//| use case:
//| Three variables are specified for historical access. 
//| Every three seconds their values should be updated to data storage for one second long.
PROGRAM PRG_HA_MultipleNodes
VAR CONSTANT
	// These connection and namespace settings need to be adapted to the runtime environment
	cOpcUaServerUrl			: STRING(MAX_STRING_LENGTH) := 'opc.tcp://localhost:4840';
	cNamespaceUri			: STRING(MAX_STRING_LENGTH) := 'urn:BeckhoffAutomation:Ua:PLC1';
END_VAR
VAR
	// Variables for HistorcalAccess
	{attribute 'OPC.UA.DA' := '1'}
	nMyValue1 : INT;	
	{attribute 'OPC.UA.DA' := '1'}
	nMyValue2 : INT;
	{attribute 'OPC.UA.DA' := '1'}
	fMyValue3 : LREAL;
	
	// state machine declarations 
	nState					: INT;
	bStart					: BOOL;  		//Set True to start this sample.
	bSample					: BOOL;			//Set True to stop the sampling.
	bStop					: BOOL;			//Set True to close the connection afterwards.
	bError					: BOOL;
	nErrorID				: DWORD;
	fbTimer					: TON:=(PT:=T#3S);
	
	// Declarations for UA_Connect
	fbUAConnect				: UA_Connect;
	stSessionConnectInfo 	: ST_UASessionConnectInfo;
	nConnectionHdl			: DWORD;
	
	// Declarations for UA_GetNamespaceIndex
	fbUAGetNamespaceIndex	: UA_GetNamespaceIndex;
	nNamespaceIndex			: UINT;
	
	// Declarations for UA_HistoryUpdate
	fbHistoryUpdateNode1	: FB_HistoryUpdate_INT := (sNodeIdentifier := 'PRG_HA_MultipleNodes.nMyValue1');
	fbHistoryUpdateNode2	: FB_HistoryUpdate_INT := (sNodeIdentifier := 'PRG_HA_MultipleNodes.nMyValue2');
	fbHistoryUpdateNode3	: FB_HistoryUpdate_LREAL := (sNodeIdentifier := 'PRG_HA_MultipleNodes.fMyValue3');
	
	// Declarations for UA_Disconnect
	fbUADisconnect			: UA_Disconnect;
	
END_VAR

nMyValue1 := nMyValue1 + 1;
nMyValue2 := nMyValue2 + 2;
fMyValue3 := fMyValue3 + 1.5;

CASE nState OF
0:	//Idle
	IF bStart THEN
		bStart				:= FALSE;
		bError				:= FALSE;
		nErrorID			:= 0;

		stSessionConnectInfo.tConnectTimeout 		:= T#1M;
		stSessionConnectInfo.tSessionTimeout 		:= T#1M;
		stSessionConnectInfo.sApplicationName		:= '';
		stSessionConnectInfo.eSecurityMode 			:= eUASecurityMsgMode_None;
		stSessionConnectInfo.eSecurityPolicyUri 	:= eUASecurityPolicy_None;
		stSessionConnectInfo.eTransportProfileUri	:= eUATransportProfileUri_UATcp;
		
		nState := 1;
	END_IF

1: //Open UA Session
	fbUAConnect(	Execute 			:= TRUE,
					ServerUrl			:= cOpcUaServerUrl,
					SessionConnectInfo	:= stSessionConnectInfo,
					Timeout				:= T#5S,
					ConnectionHdl 		=> nConnectionHdl );
		
	IF NOT fbUAConnect.Busy THEN
		IF NOT fbUAConnect.Error THEN
			nState 			:= 2;
		ELSE
			bError 			:= TRUE;
			nErrorID		:= fbUAConnect.ErrorID;
			nConnectionHdl 	:= 0;
			nState 			:= 0; //Idle
		END_IF
		fbUAConnect(Execute := FALSE);
	END_IF

2: //Get NS Index
	fbUAGetNamespaceIndex(	Execute 			:= TRUE,
							ConnectionHdl		:= nConnectionHdl,
							NamespaceUri		:= cNamespaceUri,
							NamespaceIndex		=> nNamespaceIndex );
		
	IF NOT fbUAGetNamespaceIndex.Busy THEN
		IF NOT fbUAGetNamespaceIndex.Error THEN
			nState 			:= 3;
		ELSE
			bError 			:= TRUE;
			nErrorID		:= fbUAGetNamespaceIndex.ErrorID;
			nState			:= 6; //Close Connection
		END_IF
		fbUAGetNamespaceIndex(Execute := FALSE);
	END_IF

3: //Get Node Handle & HistoryUpdate & ReleaseHandle
	//every three seconds the values should be updated for one second long.
	fbTimer(IN:=TRUE);
	IF fbTimer.ET > T#2S THEN
		bSample := TRUE;
	END_IF
	IF fbTimer.Q THEN
		bSample :=FALSE;
		fbTimer(IN:=FALSE);
	END_IF

	fbHistoryUpdateNode1(	bSample:=bSample, bStop:=bStop,	
							nConnectionHdl:=nConnectionHdl, 
							nNamespaceIndex:=nNamespaceIndex, 
							pValue:=ADR(nMyValue1) );
	IF fbHistoryUpdateNode1.bError THEN
		bError 		:= TRUE;
		nErrorID 	:= fbHistoryUpdateNode1.nErrorID;		
	END_IF

	fbHistoryUpdateNode2(	bSample:=bSample, bStop:=bStop,
							nConnectionHdl:=nConnectionHdl, 
							nNamespaceIndex:=nNamespaceIndex, 
							pValue:=ADR(nMyValue2) );
	IF fbHistoryUpdateNode2.bError THEN
		bError 		:= TRUE;
		nErrorID 	:= fbHistoryUpdateNode2.nErrorID;		
	END_IF
	
	fbHistoryUpdateNode3(	bSample:=bSample, bStop:=bStop,
							nConnectionHdl:=nConnectionHdl, 
							nNamespaceIndex:=nNamespaceIndex, 
							pValue:=ADR(fMyValue3) );
	IF fbHistoryUpdateNode2.bError THEN
		bError 		:= TRUE;
		nErrorID 	:= fbHistoryUpdateNode3.nErrorID;		
	END_IF	
	
	IF bStop 	AND NOT fbHistoryUpdateNode1.bBusy AND fbHistoryUpdateNode1.nNodeHdl = 0
				AND NOT fbHistoryUpdateNode2.bBusy AND fbHistoryUpdateNode2.nNodeHdl = 0
				AND NOT fbHistoryUpdateNode3.bBusy AND fbHistoryUpdateNode3.nNodeHdl = 0 THEN
		bStop := FALSE;
		nState := 6; //Close Connection
	END_IF 
	
6: //Close Session
	fbUADisconnect( Execute := TRUE, ConnectionHdl := nConnectionHdl );
		
	IF NOT fbUADisconnect.Busy THEN
		IF fbUAConnect.Error THEN
			bError 			:= TRUE;
			nErrorID 		:= fbUAConnect.ErrorID;
			nConnectionHdl 	:= 0;
		END_IF
		fbUAConnect(Execute := FALSE);
		nState := 0; //Idle
	END_IF
	
END_CASE

END_PROGRAM

(* stored: Version 1.1.0.1, ProductVersion 3.1.4023.6
   POU PRG_HA_MultipleNodes: Id {1c251f81-fb97-45a3-93bf-c22653fc773c}, SpecialFunc None *)
